{attribute addProperty BoxType "APS1003-7000-0016"}
{attribute addProperty Id "YVR_InputsAT %I*YVR_Inputs_32B3017D784980YVR_OutputsAT %Q*YVR_Outputs_0CD1622111681460WcStateAT %I*WcState_98A4DF7520.250InfoDataAT %I*InfoData_0BDED7BF144180"}
{attribute addProperty CRC "271105188"}
{attribute addProperty SizeInBites "2098"}
{attribute addProperty SizeInBytes "262.25"}
TYPE APS1003_D6441620 :
STRUCT
	{attribute addProperty Name "YVR_Inputs"}
	YVR_Inputs : YVR_Inputs_32B3017D;
	{attribute addProperty Name "YVR_Outputs"}
	YVR_Outputs : YVR_Outputs_0CD16221;
	{attribute addProperty Name "WcState"}
	WcState : WcState_98A4DF75;
	{attribute addProperty Name "InfoData"}
	InfoData : InfoData_0BDED7BF;
END_STRUCT
END_TYPE

(* stored: Version 1.2.0.0, ProductVersion 3.1.4024.9
   DUT APS1003_D6441620: Id {d60d8777-4e24-4542-80e3-5aa040a246fb} *)
